{attribute 'linkalways'} 
{attribute 'no_explicit_call' := 'This FB is a CLASS and must be accessed using methods or properties'}
{attribute 'enable_dynamic_creation'}
FUNCTION_BLOCK Node_F_VN_RemapImageToLogPolarSpace EXTENDS VisionNode
VAR
    ipSrcImage : _ITcVnImage;
    ipDestImage : _ITcVnImage;
    aCenter : _TcVnPoint2_REAL;
    hrPrev : _HRESULT(S_OK);
	hresult : _HRESULT(S_OK);
END_VAR

METHOD PUBLIC  Clone : I_Node
VAR
	pNode : POINTER TO Node_F_VN_RemapImageToLogPolarSpace;
END_VAR
pNode := __NEW(Node_F_VN_RemapImageToLogPolarSpace);
Clone := pNode^;
END_METHOD

METHOD FB_init : BOOL
VAR_INPUT
	bInitRetains : BOOL; // if TRUE, the retain variables are initialized (warm start / cold start)
	bInCopyCode : BOOL;  // if TRUE, the instance afterwards gets moved into the copy code (online change)
END_VAR
AddInput('ipSrcImage', ipSrcImage);
AddInput('aCenter', aCenter);
AddInput('hrPrev', hrPrev);
AddOutput('ipDestImage', ipDestImage);
AddOutput('hresult',hresult);
END_METHOD

METHOD PROTECTED OnExecute
hresult.Value := F_VN_RemapImageToLogPolarSpace(
    ipSrcImage := ipSrcImage.Value,
	ipDestImage := ipDestImage.Value,
    aCenter := aCenter.Value,
	hrPrev:= hrPrev.Value);
END_METHOD

METHOD PUBLIC PreExecutionCheck
VAR_INPUT
	Check : I_PreExecutionChecks;
END_VAR
Check.IsTrue(ipSrcImage.IsValid, 'ipSrcImage must contain an image');
END_METHOD

END_FUNCTION_BLOCK

(* stored: Version 1.1.0.1, ProductVersion 3.1.4024.13
   POU Node_F_VN_RemapImageToLogPolarSpace: Id {68396caa-f2b3-0d25-1769-d0700aa2cc6c}, SpecialFunc None
   Folder Constructor: Id {d7e7572c-7b0b-0883-044d-41d1538ddc34}
   Method Clone: Id {fc656994-ceca-0b2d-05ec-6022daa227c1}
   Method FB_init: Id {82b28ffd-fdfd-01e3-19ad-ca88a8b3ff8d}
   Method OnExecute: Id {3f362150-0004-03f1-2e6b-06435cb86711}
   Method PreExecutionCheck: Id {9968a203-7476-02ae-0f27-ee03a24b083b} *)
